// SIMATIC S7-200 project (STEP 7-Micro/WIN), CPU 224XP REL 02.01

SYMBOL_TABLE USUARIO1
P_PARO           I0.0
P_MARCHA         I0.1
LED_PARO         Q0.0
VL_U1V1W1        Q0.1
VR_U2V2W2        Q0.2
VR_CORTOCIRQUITADO Q0.3
LED_MARCHA       Q0.4
LED_AVERIA       Q0.5
END_SYMBOL_TABLE

ORGANIZATION_BLOCK PRINCIPAL:OB1
TITLE=COMENTARIOS DEL PROGRAMA
BEGIN
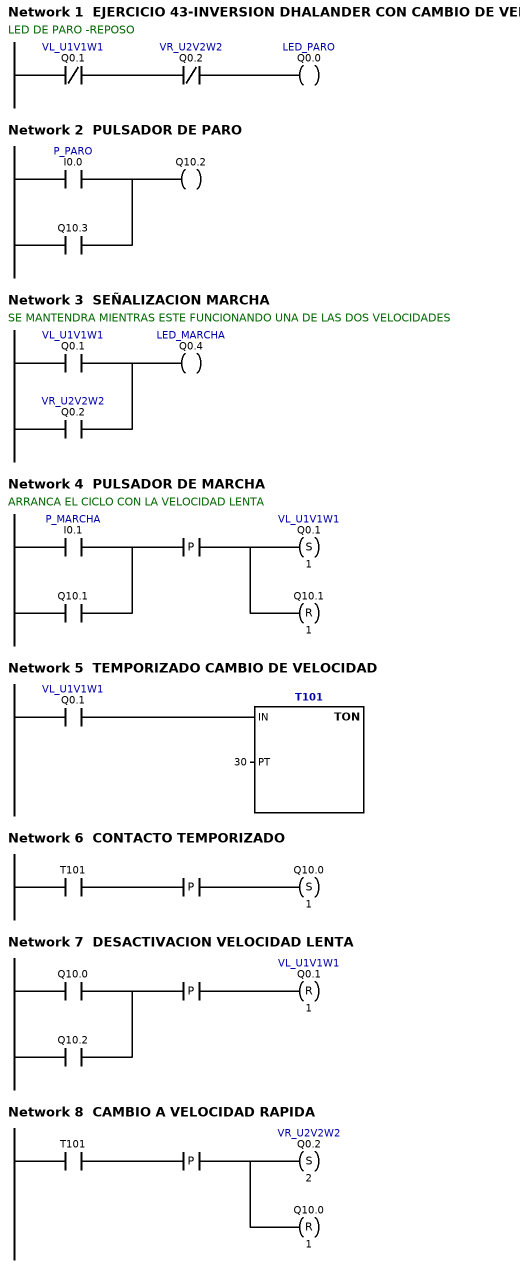
Network 1 // EJERCICIO 43-INVERSION DHALANDER CON CAMBIO DE VELOCIDAD TEMPORIZADA
// LED DE PARO -REPOSO
LDN    VL_U1V1W1:Q0.1
AN     VR_U2V2W2:Q0.2
=      LED_PARO:Q0.0
Network 2 // PULSADOR DE PARO
LD     P_PARO:I0.0
O      Q10.3
=      Q10.2
Network 3 // SEÑALIZACION MARCHA
// SE MANTENDRA MIENTRAS ESTE FUNCIONANDO UNA DE LAS DOS VELOCIDADES
LD     VL_U1V1W1:Q0.1
O      VR_U2V2W2:Q0.2
=      LED_MARCHA:Q0.4
Network 4 // PULSADOR DE MARCHA
// ARRANCA EL CICLO CON LA VELOCIDAD LENTA
LD     P_MARCHA:I0.1
O      Q10.1
EU
S      VL_U1V1W1:Q0.1, 1
R      Q10.1, 1
Network 5 // TEMPORIZADO CAMBIO DE VELOCIDAD
LD     VL_U1V1W1:Q0.1
TON    T101, 30
Network 6 // CONTACTO TEMPORIZADO 
LD     T101
EU
S      Q10.0, 1
Network 7 // DESACTIVACION VELOCIDAD LENTA
LD     Q10.0
O      Q10.2
EU
R      VL_U1V1W1:Q0.1, 1
Network 8 // CAMBIO A VELOCIDAD RAPIDA
LD     T101
EU
S      VR_U2V2W2:Q0.2, 2
R      Q10.0, 1
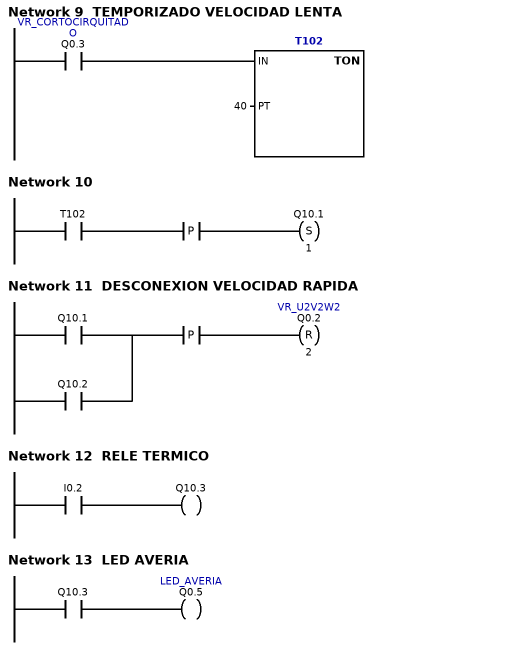
Network 9 // TEMPORIZADO VELOCIDAD LENTA 
LD     VR_CORTOCIRQUITADO:Q0.3
TON    T102, 40
Network 10
LD     T102
EU
S      Q10.1, 1
Network 11 // DESCONEXION VELOCIDAD RAPIDA
LD     Q10.1
O      Q10.2
EU
R      VR_U2V2W2:Q0.2, 2
Network 12 // RELE TERMICO
LD     I0.2
=      Q10.3
Network 13 // LED AVERIA
LD     Q10.3
=      LED_AVERIA:Q0.5
END_ORGANIZATION_BLOCK
